// TIA Portal project "Lezione1_CorsoBase" (V19)

(* hardware
DEVICE "S7-1200 station_1"  S7-1200 Station
   slot 0: "Rack_0"  S7-1200 Rack  Rack  V1.0
   slot 1: "PLC_1"  CPU 1214C AC/DC/Rly  6ES7 214-1BG40-0XB0  V4.1
*)

// ===== PLC "PLC_1"  CPU 1214C AC/DC/Rly =====

VAR_GLOBAL   // PLC tag table "Default tag table"
   "PulsanteEmergenza" AT %I0.0 : Bool;
   "PulsanteStop" AT %I0.1 : Bool;
   "TermicaMotore" AT %I0.2 : Bool;
   "StartAvanti" AT %I0.3 : Bool;
   "StartIndietro" AT %I0.4 : Bool;
   "ResetAllarmi" AT %I0.5 : Bool;
   "ResetConteggio" AT %I0.6 : Bool;
   "MotoreAvanti" AT %Q0.0 : Bool;
   "MotoreIndietro" AT %Q0.1 : Bool;
   "LampadaVerde" AT %Q0.2 : Bool;
   "LampadaGialla" AT %Q0.3 : Bool;
   "LampadaRossa" AT %Q0.4 : Bool;
END_VAR

ORGANIZATION_BLOCK "Main"   // OB1, LAD, ProgramCycle
TITLE = "Main Program Sweep (Cycle)"
{ S7_Optimized_Access := 'TRUE' }
VERSION : 0.1
   VAR_INPUT
      Initial_Call : Bool;   // Initial call of this OB
      Remanence : Bool;   // =True, if remanent data are available
   END_VAR
BEGIN

REGION Network 1
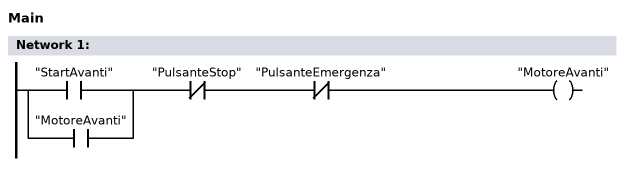
   RUNG wire#powerrail
      Contact( "StartAvanti" )
      wire#w1
      I_Contact( "PulsanteStop" )
      I_Contact( "PulsanteEmergenza" )
      Coil( "MotoreAvanti" )
   END_RUNG
   RUNG wire#powerrail
      Contact( "MotoreAvanti" )
   END_RUNG wire#w1
   // the same network as SCL:
   "MotoreAvanti" := ("StartAvanti" OR "MotoreAvanti") AND NOT "PulsanteStop" AND NOT "PulsanteEmergenza";
END_REGION
END_ORGANIZATION_BLOCK